TYPE ST_HMI_Monitor_CoolingSystem :
STRUCT
	e_OperationMode 		: eCoolingSystemState;
	e_HeatPumpStatus		: eHeatPumpState;
	r_CoolantTemperature	:	REAL;
	r_CoolantPressure		:	REAL;
	r_EnclosureDewpoint		:	REAL;
	b_HeatPumpError			: 	BOOL;
	b_HeatPumpWarning		:	BOOL;
	b_CoolantPressureWarning: 	BOOL;
	b_CoolantPressureError	:	BOOL;
	b_CoolantTempWarning	: 	BOOL;
END_STRUCT
END_TYPE

(* stored: Version 1.1.0.1, ProductVersion 3.1.4026.18
   DUT ST_HMI_Monitor_CoolingSystem: Id {bc8b2866-8d72-4ede-b742-b1d817d7c9ea} *)
